KUKA KRL data list: Thay_Mo.dat

&ACCESS RV
&REL 1
DEFDAT Thay_Mo PUBLIC
  DECL E6POS HOME={A1 0.0, A2 -90.0, A3 90.0, A4 0.0, A5 0.0, A6 0.0}
  DECL E6POS P_GREASE={X 200.0, Y 0.0, Z 800.0, A 0.0, B 0.0, C 0.0, S 2, T 10}
ENDDAT
